// TIA Portal V20 export
DATA_BLOCK "SBK13"   // DB327
// stored: MemoryReserve 100
   VAR
      "SAFETY DOOR LOCK10.INPUT" : Bool := FALSE;
      SPARE : Bool := FALSE;
      "SAFETY DOOR LOCK12.INPUT" : Bool := FALSE;
      SPARE_1 : Bool := FALSE;
      "SAFETY DOOR LOCK10.INPUT_1" : Bool := FALSE;
      SPARE_2 : Bool := FALSE;
      "SAFETY DOOR LOCK12.INPUT_1" : Bool := FALSE;
      SPARE_3 : Bool := FALSE;
      "SAFETY DOOR LOCK10.OUTPUT" : Bool := FALSE;
      SPARE_4 : Bool := FALSE;
      "SAFETY DOOR LOCK12.OUTPUT" : Bool := FALSE;
   END_VAR
BEGIN
END_DATA_BLOCK
